Fanuc KAREL source: kt00547.KL

-- PROVISIONAL review KL for V770-1; original PC SHA256 a564cf70c8b663e46fd370eda81a90cef342873f2ef9856493c42c4a89195420
-- Incomplete behavior may be omitted. Consult companion uncertainty JSON. Do not deploy.
PROGRAM KT00547
%NOLOCKGROUP
-- UNRESOLVED_DECL P1 type=000199
-- UNRESOLVED_DECL P2 type=000106
-- UNRESOLVED_DECL OUT type=000199
BEGIN
  -- UNRESOLVED_PC offsets 5-20; opcodes 2E,22,32,35
  -- UNRESOLVED_PC offsets 25-64; opcodes 49,7E,49,7E,60,7E,4A
  -- UNRESOLVED_PC offsets 69-73; opcodes 7F
END KT00547
